PROGRAM prgFileHnd
VAR
	bWrite			: BOOL := FALSE;(* Rising edge starts program execution *)
	sNetId			: T_AmsNetId := '';	(* TwinCAT system network address *)
	sFileName		: T_MaxString := 'MyFile';(* CSV destination file path and name *)
	bError			: BOOL;
	nErrId			: UDINT;
	hFile			: UINT		:= 0;(* File handle of the source file *)
	step			: DWORD 	:= 0;

	fbFileOpen	: FB_FileOpen;(* Opens file *)
	fbFileClose	: FB_FileClose;(* Closes file *)
	fbFileWrite	: FB_FileWrite;(* Reads binary data *)	
	trig:R_trig;
	sErr: STRING;
	sMsg: STRING;
	
	//Read
	bRead: BOOL;
	sFileNameRead:T_MaxString;
	bErrorRead:BOOL;
	nErrIdRead:UDINT;
	stepRead:UINT;
	hFileRead:UINT;
	trigRead:R_TRIG;
	
	fbFileOpenRead	: FB_FileOpen;(* Opens file *)
	fbFileCloseRead	: FB_FileClose;(* Closes file *)
	fbFileRead	: FB_FileRead;(* Reads binary data *)
	
	sMsgRead: STRING;
	sErrRead: STRING;
//	sFilePath:T_MaxString:='C:\Relat\';
	sFullfileName: T_MaxString;
END_VAR

trig(CLK:= bWrite);

CASE step OF 
	0:
		IF trig.Q THEN
			step:=10;
			fbFileOpen(bExecute:= FALSE);
			fbFileClose(bExecute:= FALSE);
			fbFileWrite(bExecute:= FALSE);
			sMsg:='Abrindo arquivo';
			sErr:='';
		END_IF
	10:
		sFullfileName:= concat(prgFileManipulation.path, concat(concat('\', sFileName),'.bkp'));
		fbFileOpen(sNetId:=sNetId , sPathName:= sFullfileName, nMode:= FOPEN_MODEWRITE OR FOPEN_MODEBINARY, 
			ePath:= PATH_GENERIC, bExecute:= TRUE, tTimeout:= T#10S, bError => bError, nErrId => nErrId);
		IF NOT fbFileOpen.bBusy THEN
			IF NOT fbFileOpen.bError THEN
				step:=20;
				hFile:= fbFileOpen.hFile;
				sMsg:='Escrevendo arquivo';
			ELSE
				step:=100;
				sErr:='Erro ao abrir o arquivo';
			END_IF
		END_IF
	20:
		fbFileWrite(sNetId:= sNetId, hFile:= hFile,	pWriteBuff:=ADR(main.aStructs), cbWriteLen:= SIZEOF(MAIN.aStructs),
			bExecute:= TRUE,tTimeout:=T#20S, bError => bError, nErrId => nErrId);
		IF NOT fbFileWrite.bBusy THEN
			IF NOT fbFileWrite.bError THEN
				step:=30;
				sMsg:='Arquivo salvo';
			ELSE
				step:=100;
				sErr:='Erro ao escrever o arquivo';	
			END_IF
		END_IF
	30:
		fbFileClose( sNetId := sNetId, hFile := hFile, bExecute := TRUE, bError => bError, nErrId => nErrId);
		IF NOT fbFileClose.bBusy THEN
			step:=100;
			hFile:=0;
			GVL.updateFileList:=TRUE;
		END_IF
	100:
		IF hFile <> 0 THEN
			step:=30;
		ELSE
			step:=0;
			sMsg:='';
		END_IF
END_CASE

trigRead(CLK:= bRead);
CASE stepRead OF
	0:
		IF trigRead.Q THEN
			stepRead:=10;
			fbFileOpenRead(bExecute:= FALSE);
			fbFileCloseRead(bExecute:= FALSE);
			fbFileRead(bExecute:= FALSE);
			sMsgRead:='Abrindo arquivo';
			sErrRead:='';
		END_IF
	10:
		sFileNameRead:= concat(prgFileManipulation.path, concat('\',prgFileManipulation.selectedLocalFile));
		fbFileOpenRead(sNetId:=sNetId , sPathName:= sFileNameRead, nMode:= FOPEN_MODEREAD OR FOPEN_MODEBINARY, 
			ePath:= PATH_GENERIC, bExecute:= TRUE, tTimeout:= T#10S, bError => bErrorRead, nErrId => nErrIdRead);
		IF NOT fbFileOpenRead.bBusy THEN
			IF NOT fbFileOpenRead.bError THEN
				hFileRead:= fbFileOpenRead.hFile;
				stepRead:=20;
			ELSE
				stepRead:=100;	
				sErrRead:='Erro ao abrir arquivo para leitura';
			END_IF
		END_IF
	20:
		fbFileRead(sNetId:=sNetId ,hFile:=hFileRead ,pReadBuff:=ADR(MAIN.aStructs) ,cbReadLen:=SIZEOF(MAIN.aStructs) ,bExecute:=TRUE , 
			tTimeout:= T#30S,bError=> bErrorRead, nErrId=>nErrIdRead);
		IF NOT fbFileRead.bBusy THEN
			IF NOT fbFileRead.bError THEN
				stepRead:=30;
			ELSE
				stepRead:=100;
				sErrRead:='Erro ao ler o arquivo';
			END_IF
		END_IF
	30:
		fbFileCloseRead( sNetId := sNetId, hFile := hFileRead, bExecute := TRUE, bError => bErrorRead, nErrId => nErrIdRead);
		IF NOT fbFileCloseRead.bBusy THEN
			stepRead:=100;
			hFileRead:=0;
			GVL.updateFileList:=TRUE;
		END_IF
	100:
		IF hFileRead <> 0 THEN
			stepRead:=30;
		ELSE
			stepRead:=0;
			sMsgRead:='';
		END_IF
END_CASE

END_PROGRAM

(* stored: Version 1.1.0.1, ProductVersion 3.1.4024.12
   POU prgFileHnd: Id {faefe0c5-7146-4765-a57a-913fd07e3fa3}, SpecialFunc None *)
